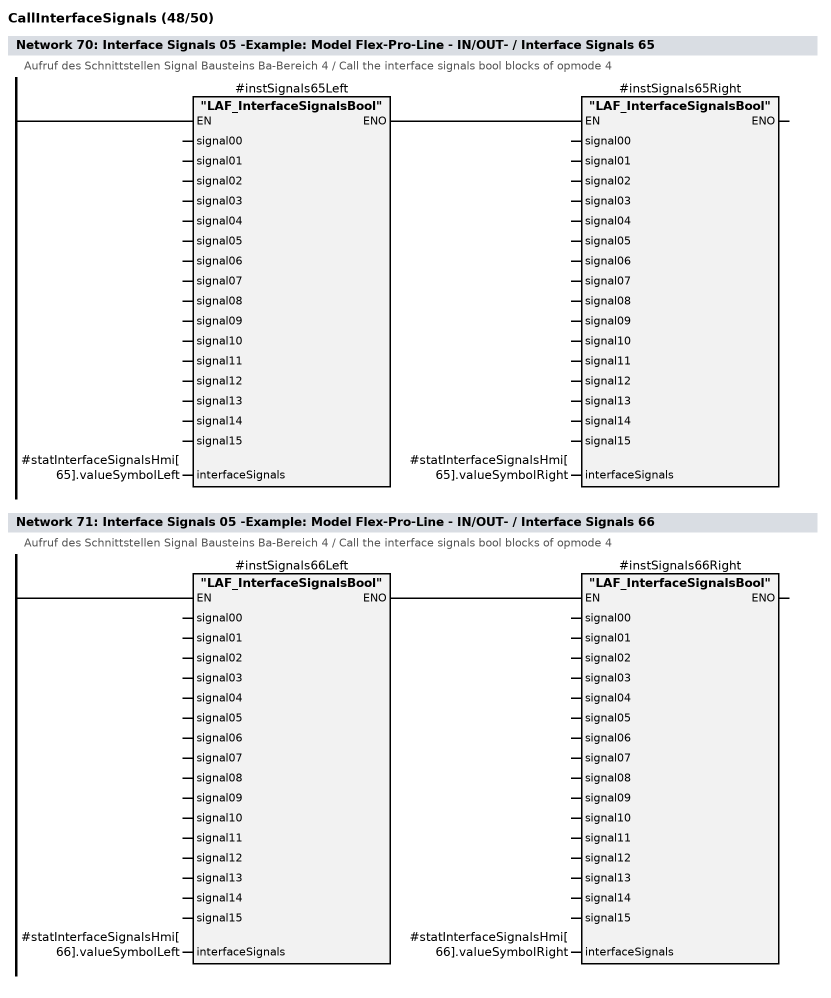
   RUNG wire#powerrail
      #instSignals65Left(signal00 :=, signal01 :=, signal02 :=, signal03 :=, signal04 :=, signal05 :=, signal06 :=, signal07 :=, signal08 :=, signal09 :=, signal10 :=, signal11 :=, signal12 :=, signal13 :=, signal14 :=, signal15 :=, interfaceSignals := #statInterfaceSignalsHmi[65].valueSymbolLeft)
      #instSignals65Right(signal00 :=, signal01 :=, signal02 :=, signal03 :=, signal04 :=, signal05 :=, signal06 :=, signal07 :=, signal08 :=, signal09 :=, signal10 :=, signal11 :=, signal12 :=, signal13 :=, signal14 :=, signal15 :=, interfaceSignals := #statInterfaceSignalsHmi[65].valueSymbolRight)
   END_RUNG
   // the same network as SCL:
   #instSignals65Left(interfaceSignals := #statInterfaceSignalsHmi[65].valueSymbolLeft, ENO => #_w1);   // "LAF_InterfaceSignalsBool"
   IF #_w1 THEN
       #instSignals65Right(interfaceSignals := #statInterfaceSignalsHmi[65].valueSymbolRight);   // "LAF_InterfaceSignalsBool"
   END_IF;
END_REGION

REGION Network 71: Interface Signals 05 -Example: Model Flex-Pro-Line - IN/OUT- / Interface Signals 66
   // Aufruf des Schnittstellen Signal Bausteins Ba-Bereich 4 / Call the interface signals bool blocks of opmode 4
   RUNG wire#powerrail
      #instSignals66Left(signal00 :=, signal01 :=, signal02 :=, signal03 :=, signal04 :=, signal05 :=, signal06 :=, signal07 :=, signal08 :=, signal09 :=, signal10 :=, signal11 :=, signal12 :=, signal13 :=, signal14 :=, signal15 :=, interfaceSignals := #statInterfaceSignalsHmi[66].valueSymbolLeft)
      #instSignals66Right(signal00 :=, signal01 :=, signal02 :=, signal03 :=, signal04 :=, signal05 :=, signal06 :=, signal07 :=, signal08 :=, signal09 :=, signal10 :=, signal11 :=, signal12 :=, signal13 :=, signal14 :=, signal15 :=, interfaceSignals := #statInterfaceSignalsHmi[66].valueSymbolRight)
   END_RUNG
   // the same network as SCL:
   #instSignals66Left(interfaceSignals := #statInterfaceSignalsHmi[66].valueSymbolLeft, ENO => #_w1);   // "LAF_InterfaceSignalsBool"
   IF #_w1 THEN
       #instSignals66Right(interfaceSignals := #statInterfaceSignalsHmi[66].valueSymbolRight);   // "LAF_InterfaceSignalsBool"
   END_IF;
END_REGION

REGION Network 72: Interface Signals 05 -Example: Model Flex-Pro-Line - IN/OUT- / Interface Signals 67
   // Aufruf des Schnittstellen Signal Bausteins Ba-Bereich 4 / Call the interface signals bool blocks of opmode 4
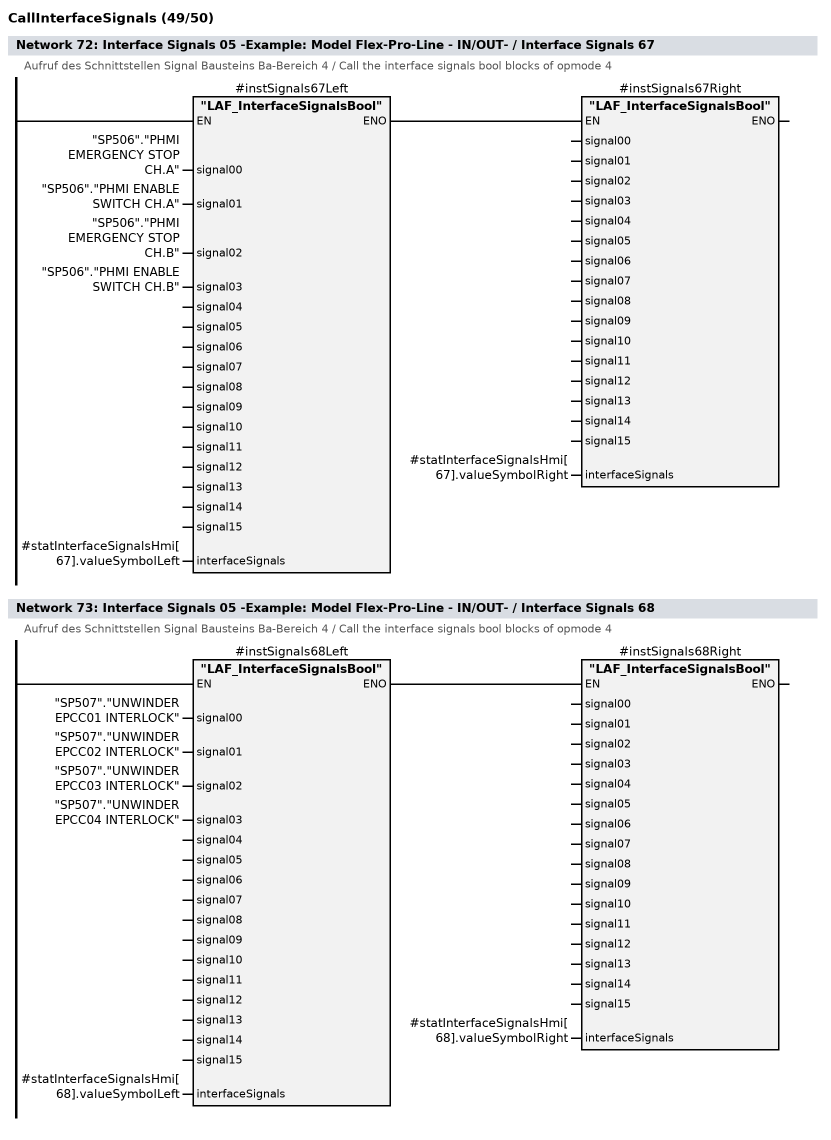
   RUNG wire#powerrail
      #instSignals67Left(signal00 := "SP506"."PHMI EMERGENCY STOP CH.A", signal01 := "SP506"."PHMI ENABLE SWITCH CH.A", signal02 := "SP506"."PHMI EMERGENCY STOP CH.B", signal03 := "SP506"."PHMI ENABLE SWITCH CH.B", signal04 :=, signal05 :=, signal06 :=, signal07 :=, signal08 :=, signal09 :=, signal10 :=, signal11 :=, signal12 :=, signal13 :=, signal14 :=, signal15 :=, interfaceSignals := #statInterfaceSignalsHmi[67].valueSymbolLeft)
      #instSignals67Right(signal00 :=, signal01 :=, signal02 :=, signal03 :=, signal04 :=, signal05 :=, signal06 :=, signal07 :=, signal08 :=, signal09 :=, signal10 :=, signal11 :=, signal12 :=, signal13 :=, signal14 :=, signal15 :=, interfaceSignals := #statInterfaceSignalsHmi[67].valueSymbolRight)
   END_RUNG
   // the same network as SCL:
   #instSignals67Left(signal00 := "SP506"."PHMI EMERGENCY STOP CH.A",   // "LAF_InterfaceSignalsBool"
                      signal01 := "SP506"."PHMI ENABLE SWITCH CH.A",
                      signal02 := "SP506"."PHMI EMERGENCY STOP CH.B",
                      signal03 := "SP506"."PHMI ENABLE SWITCH CH.B",
                      interfaceSignals := #statInterfaceSignalsHmi[67].valueSymbolLeft,
                      ENO => #_w1);
   IF #_w1 THEN
       #instSignals67Right(interfaceSignals := #statInterfaceSignalsHmi[67].valueSymbolRight);   // "LAF_InterfaceSignalsBool"
   END_IF;
END_REGION

REGION Network 73: Interface Signals 05 -Example: Model Flex-Pro-Line - IN/OUT- / Interface Signals 68
   // Aufruf des Schnittstellen Signal Bausteins Ba-Bereich 4 / Call the interface signals bool blocks of opmode 4
   RUNG wire#powerrail
      #instSignals68Left(signal00 := "SP507"."UNWINDER EPCC01 INTERLOCK", signal01 := "SP507"."UNWINDER EPCC02 INTERLOCK", signal02 := "SP507"."UNWINDER EPCC03 INTERLOCK", signal03 := "SP507"."UNWINDER EPCC04 INTERLOCK", signal04 :=, signal05 :=, signal06 :=, signal07 :=, signal08 :=, signal09 :=, signal10 :=, signal11 :=, signal12 :=, signal13 :=, signal14 :=, signal15 :=, interfaceSignals := #statInterfaceSignalsHmi[68].valueSymbolLeft)
      #instSignals68Right(signal00 :=, signal01 :=, signal02 :=, signal03 :=, signal04 :=, signal05 :=, signal06 :=, signal07 :=, signal08 :=, signal09 :=, signal10 :=, signal11 :=, signal12 :=, signal13 :=, signal14 :=, signal15 :=, interfaceSignals := #statInterfaceSignalsHmi[68].valueSymbolRight)
   END_RUNG
   // the same network as SCL:
   #instSignals68Left(signal00 := "SP507"."UNWINDER EPCC01 INTERLOCK",   // "LAF_InterfaceSignalsBool"
                      signal01 := "SP507"."UNWINDER EPCC02 INTERLOCK",
                      signal02 := "SP507"."UNWINDER EPCC03 INTERLOCK",
                      signal03 := "SP507"."UNWINDER EPCC04 INTERLOCK",
                      interfaceSignals := #statInterfaceSignalsHmi[68].valueSymbolLeft,
                      ENO => #_w1);
   IF #_w1 THEN
       #instSignals68Right(interfaceSignals := #statInterfaceSignalsHmi[68].valueSymbolRight);   // "LAF_InterfaceSignalsBool"
   END_IF;
END_REGION

REGION Network 74: Interface Signals 05 -Example: Model Flex-Pro-Line - IN/OUT- / Interface Signals 69
   // Aufruf des Schnittstellen Signal Bausteins Ba-Bereich 4 / Call the interface signals bool blocks of opmode 4
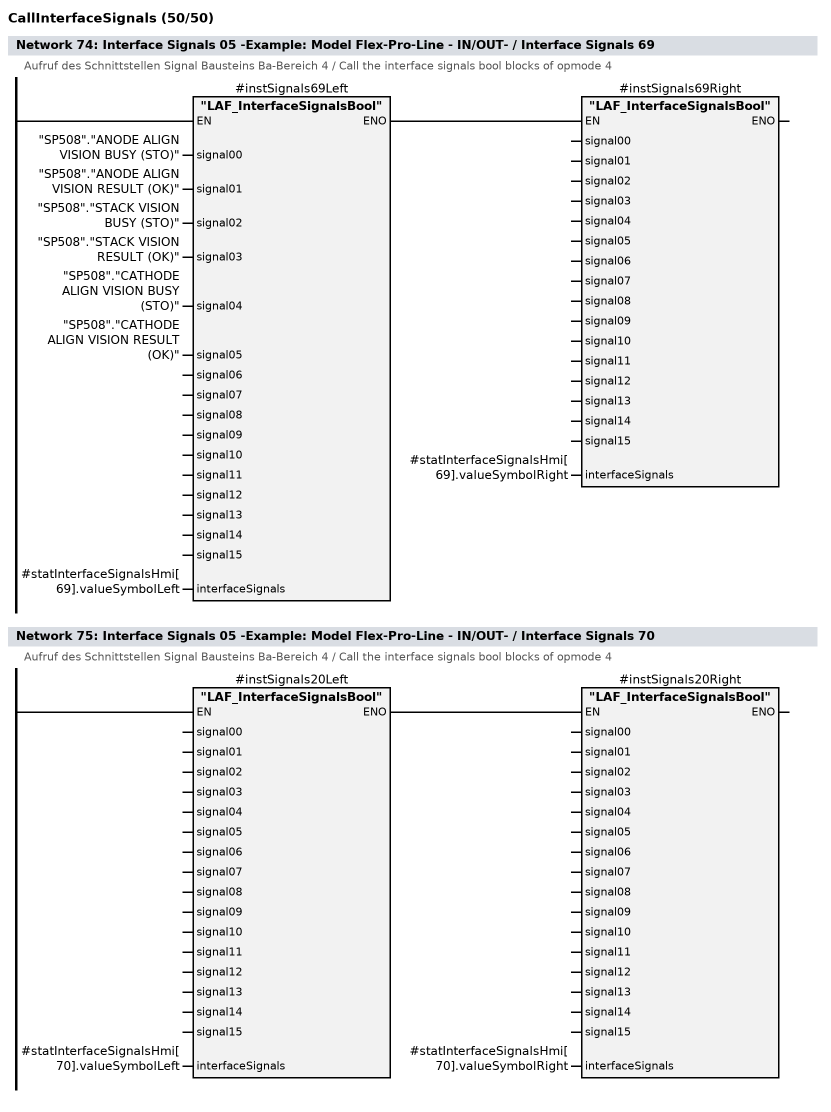
   RUNG wire#powerrail
      #instSignals69Left(signal00 := "SP508"."ANODE ALIGN VISION BUSY (STO)", signal01 := "SP508"."ANODE ALIGN VISION RESULT (OK)", signal02 := "SP508"."STACK VISION BUSY (STO)", signal03 := "SP508"."STACK VISION RESULT (OK)", signal04 := "SP508"."CATHODE ALIGN VISION BUSY (STO)", signal05 := "SP508"."CATHODE ALIGN VISION RESULT (OK)", signal06 :=, signal07 :=, signal08 :=, signal09 :=, signal10 :=, signal11 :=, signal12 :=, signal13 :=, signal14 :=, signal15 :=, interfaceSignals := #statInterfaceSignalsHmi[69].valueSymbolLeft)
      #instSignals69Right(signal00 :=, signal01 :=, signal02 :=, signal03 :=, signal04 :=, signal05 :=, signal06 :=, signal07 :=, signal08 :=, signal09 :=, signal10 :=, signal11 :=, signal12 :=, signal13 :=, signal14 :=, signal15 :=, interfaceSignals := #statInterfaceSignalsHmi[69].valueSymbolRight)
   END_RUNG
   // the same network as SCL:
   #instSignals69Left(signal00 := "SP508"."ANODE ALIGN VISION BUSY (STO)",   // "LAF_InterfaceSignalsBool"
                      signal01 := "SP508"."ANODE ALIGN VISION RESULT (OK)",
                      signal02 := "SP508"."STACK VISION BUSY (STO)",
                      signal03 := "SP508"."STACK VISION RESULT (OK)",
                      signal04 := "SP508"."CATHODE ALIGN VISION BUSY (STO)",
                      signal05 := "SP508"."CATHODE ALIGN VISION RESULT (OK)",
                      interfaceSignals := #statInterfaceSignalsHmi[69].valueSymbolLeft,
                      ENO => #_w1);
   IF #_w1 THEN
       #instSignals69Right(interfaceSignals := #statInterfaceSignalsHmi[69].valueSymbolRight);   // "LAF_InterfaceSignalsBool"
   END_IF;
END_REGION

REGION Network 75: Interface Signals 05 -Example: Model Flex-Pro-Line - IN/OUT- / Interface Signals 70
   // Aufruf des Schnittstellen Signal Bausteins Ba-Bereich 4 / Call the interface signals bool blocks of opmode 4
   RUNG wire#powerrail
      #instSignals20Left(signal00 :=, signal01 :=, signal02 :=, signal03 :=, signal04 :=, signal05 :=, signal06 :=, signal07 :=, signal08 :=, signal09 :=, signal10 :=, signal11 :=, signal12 :=, signal13 :=, signal14 :=, signal15 :=, interfaceSignals := #statInterfaceSignalsHmi[70].valueSymbolLeft)
      #instSignals20Right(signal00 :=, signal01 :=, signal02 :=, signal03 :=, signal04 :=, signal05 :=, signal06 :=, signal07 :=, signal08 :=, signal09 :=, signal10 :=, signal11 :=, signal12 :=, signal13 :=, signal14 :=, signal15 :=, interfaceSignals := #statInterfaceSignalsHmi[70].valueSymbolRight)
   END_RUNG
   // the same network as SCL:
   #instSignals20Left(interfaceSignals := #statInterfaceSignalsHmi[70].valueSymbolLeft, ENO => #_w1);   // "LAF_InterfaceSignalsBool"
   IF #_w1 THEN
       #instSignals20Right(interfaceSignals := #statInterfaceSignalsHmi[70].valueSymbolRight);   // "LAF_InterfaceSignalsBool"
   END_IF;
END_REGION
END_FUNCTION_BLOCK
